Fanuc KAREL source: J_IN_RANGE.kl

PROGRAM T
%NOLOCKGROUP
VAR
 v0 : JOINTPOS
 res : BOOLEAN
BEGIN
 res = J_IN_RANGE(v0)
END T
